PROGRAM Stn054_31_Stn311MergePrestop
VAR
// correct
	{attribute 'TcLinkToOSO' := '
			.iPuckPresent  :=  <0,1,2>TIIB[N57S00 (AL1332)]^N57S01 (AL2341)^TxPDO^input byte 0;
			.iBufferFull :=  <0,1,2>TIIB[N57S00 (AL1332)]^N57S01 (AL2341)^TxPDO^input byte 2;
			.oStopLower  :=  <0,1,1>TIIB[N57S00 (AL1332)]^N57S02 (EX260)^RxPDO^output byte 0'}

	fbConvStop: FB_ConvStop;
END_VAR

//  This code instantiates a component that is implimented as a common function block
//    Note that I/O is linked directly to I/O variables inside the named instance

gStn054_31_Stn311MergePrestop.ConvRunning  := gConsumed_SafetyInterfaceConv.MtrRunning.Enc058Mtr05;

fbConvStop(
	pStn := ADR(gStn054),
	pCmp := ADR(gStn054_31_Stn311MergePrestop),
	pUpstreamStop := 0,
	pStateTraceBuffer := ADR(gStn054_StateTraceBuffer),
	pStateTraceFifo := ADR(gStn054_StateTraceFifo),
	pStats := ADR(gStn054_02_Stats));

END_PROGRAM

(* stored: Version 1.1.0.1, ProductVersion 3.1.4024.6
   POU Stn054_31_Stn311MergePrestop: Id {3a2c1ca7-ddfb-4d72-a64a-8f385c5d77f7}, SpecialFunc None *)
